// TwinCAT 3 PLC project PLC
// ProgramVersion: 3.1.4024.0
// libraries:
//   Tc2_Standard, * (Beckhoff Automation GmbH)
//   Tc2_System, * (Beckhoff Automation GmbH)
//   Tc3_Module, * (Beckhoff Automation GmbH)
// project tree:
//   / PlcTask.TcTTO
//   POUs/Course/ FN_2_2_Finite_State_Machine.TcPOU
//   POUs/ MAIN.TcPOU
// real-time tasks:
//   TASK PlcTask: cycle T#10ms, priority 20, ADS port 350

CONFIGURATION PLC
    RESOURCE PLC ON TwinCAT3
        TASK PlcTask(INTERVAL := T#10ms, PRIORITY := 20);
        PROGRAM MAIN WITH PlcTask : MAIN;
    END_RESOURCE
END_CONFIGURATION

// ---- POUs/MAIN.TcPOU
PROGRAM MAIN
VAR
	Lesson_2_2 : FN_2_2_Finite_State_Machine;
END_VAR

Lesson_2_2();

END_PROGRAM

// ---- POUs/Course/FN_2_2_Finite_State_Machine.TcPOU
FUNCTION_BLOCK FN_2_2_Finite_State_Machine

VAR CONSTANT
	MIXERDURATION : TIME := T#5S;
	PUMPDURATION  : TIME := T#3S;
	GATEDURATION  : TIME := T#2S;	
END_VAR

VAR_INPUT
	startPB : BOOL;
	stopPB : BOOL;
END_VAR

VAR_OUTPUT
	mixerState : BOOL;
	pumpState  : BOOL;
	gateState  : BOOL;
END_VAR

VAR
	startTrig : R_TRIG;
	stopTrig  : R_TRIG;

	state : (init, mixerON, pumpON, gateOpen, close);

	timer : TON;
END_VAR

stopTrig(CLK := stopPB);

IF NOT stopPB THEN // Ensure Stop PB is not pressed before checking startPB
	startTrig(CLK := startPB);
END_IF

CASE state OF
	init : // default state
		IF startTrig.Q THEN
			state := mixerON;
		END_IF
	
	mixerON: // Turn ON mixer for MIXERDURATION[default 5s]
		mixerState := TRUE;
		timer(IN := TRUE, PT := MIXERDURATION);	
		IF timer.Q THEN
			timer(IN := FALSE);
			state := pumpON;
		END_IF
	
	pumpON: // Turn ON pump for PUMPDURATION[default 4s]
		pumpState := TRUE;
		timer(IN := TRUE, PT := PUMPDURATION);	
		IF timer.Q THEN
			pumpState := FALSE;
			timer(IN := FALSE);
			state := gateOpen;
		END_IF
	
	gateOpen: // Open gate for GATEDURATION[default 3s]
		timer(IN := TRUE, PT := GATEDURATION);	
		IF timer.Q THEN
			timer(IN := FALSE);
			state := close;
		END_IF
	
	close: // Tidy up variables and loop to start
		M_resetvariables();
		state := init;
END_CASE

IF stopTrig.Q THEN
	state := close;
END_IF

METHOD PRIVATE M_resetvariables : BOOL
VAR_INPUT
END_VAR
timer(IN := FALSE);	
mixerState := FALSE;
pumpState := FALSE;
gateState := FALSE;
END_METHOD

END_FUNCTION_BLOCK
